FUNCTION_BLOCK CruiseController_FBDKTestBench (* Composite Function Block Type *)
  (* Standard: 61499-2 *)
  (* Version 0.2, 2003-12-05, JHC, Rockwell Automation, Renamed from NEWCOMPFB. *)
  (* Version 0.1, 2002-01-08, JHC, Rockwell Automation, Added DLY FB as example. *)
  (* Version 0.0, 2000-05-27, JHC, Rockwell Automation *)
  (* Compiler header: package fb.rt.benchmarks.cruisecontrol; *)
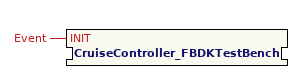
  EVENT_INPUT
    INIT; (* Initialization Request *)
  END_EVENT
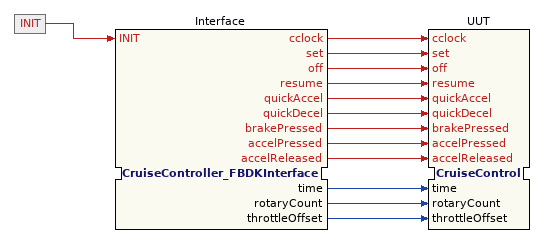
  FBS
    Interface : CruiseController_FBDKInterface;
    UUT : CruiseControl;
  END_FBS
  EVENT_CONNECTIONS
    Interface.cclock TO UUT.cclock;
    Interface.set TO UUT.set;
    Interface.off TO UUT.off;
    Interface.resume TO UUT.resume;
    Interface.quickAccel TO UUT.quickAccel;
    Interface.quickDecel TO UUT.quickDecel;
    Interface.brakePressed TO UUT.brakePressed;
    Interface.accelPressed TO UUT.accelPressed;
    Interface.accelReleased TO UUT.accelReleased;
    INIT TO Interface.INIT;
  END_CONNECTIONS
  DATA_CONNECTIONS
    Interface.time TO UUT.time;
    Interface.rotaryCount TO UUT.rotaryCount;
    Interface.throttleOffset TO UUT.throttleOffset;
  END_CONNECTIONS
END_FUNCTION_BLOCK
